TYPE ENUM_SLOT_TYPE :
(
	SETUP := 0,
	LOGIC := 1,
	TEARDOWN := 2
);
END_TYPE

(* stored: Version 1.1.0.1, ProductVersion 3.1.4024.10
   DUT ENUM_SLOT_TYPE: Id {0d1729dc-b912-42e3-ba01-dd8bc9e7f924} *)
